TYPE ST_Message :
STRUCT
  eType         : e_MessageType;
  eDevice       : e_Device;
  eSubdevice    : e_SubDevice;
  {attribute 'displaymode':='hex'}
  iErrorNumber  : LINT;
  tTime         : STRING(24);
  sText         : STRING(256);
END_STRUCT
END_TYPE

(* stored: Version 1.1.0.1, ProductVersion 3.1.4024.4
   DUT ST_Message: Id {1d190b77-cb88-4f2d-8c5f-8826899ae411} *)
